PROGRAM PRG_SharedCore
VAR
END_VAR

F_CreateCPULoad();

END_PROGRAM

(* stored: Version 1.1.0.1, ProductVersion 3.1.4026.18
   POU PRG_SharedCore: Id {89a2c607-fd4b-45ff-adb0-14a7981190a3}, SpecialFunc None *)
